FUNCTION_BLOCK MoveUp EXTENDS GuardMove
VAR_INPUT
END_VAR
VAR_OUTPUT
END_VAR
VAR
END_VAR

(*

short summary
=================
This abstract property returns the class name of the concrete object, 
which is useful for logging/debugging purpose or to check the class name
for ``__DELETE`` in factories (sometimes it's necessary to do more 
than just to free the memory).

.. <legal notes>

legal notes
=================
| SPDX-FileCopyrightText: © 2022 ekvip automation GmbH <info@ekvip.de>
| SPDX-License-Identifier: Apache-2.0
| For details check: Apache-2.0_

.. _Apache-2.0: https://www.apache.org/licenses/LICENSE-2.0

.. </legal notes>

*)
PROPERTY className : CNM_AbstractObject.ClassName
GET
className := 'MoveUp';
END_GET
END_PROPERTY

PROPERTY PROTECTED direction : Rotation
GET
direction := Rotation.UP;
END_GET
END_PROPERTY

END_FUNCTION_BLOCK

(* stored: Version 1.1.0.1
   POU MoveUp: Id {c1094bb1-d2f6-468f-93a8-56ebf9fe4836}, SpecialFunc None
   Property className: Id {f3c5538d-a1db-414c-b088-3a2b7e12f57c}
   Get Get: Id {2be7ccd5-cd9d-4e37-89cd-2c09c8176995}
   Property direction: Id {29b1c5db-12e4-4678-90b0-7c8e04f7e1b1}
   Get Get: Id {80006c31-1add-466f-ac89-742d4197a330} *)
